FUNCTION_BLOCK ModbusRTU_EM_Bell
VAR_INPUT
	MB_FirstUnitID: BYTE;
	MB_LastUnitID:  BYTE;
	EM_First: INT := 1;
END_VAR
VAR_OUTPUT
END_VAR
VAR
END_VAR

END_FUNCTION_BLOCK

(* stored: Version 1.1.0.1, ProductVersion 3.1.4024.12
   POU ModbusRTU_EM_Bell: Id {82da657d-d222-4279-baf3-7e4e6d4c96bd}, SpecialFunc None *)
